// TIA Portal project "openness_project" (V17)

(* hardware
DEVICE "S71500/ET200MP station_1"  S7-1500 station
   slot 0: "Rail_0"  Rack  6ES7 590-1***0-0AA0
   slot 1: "N0001-S1-MC1.CC1-K30001"  CPU 1515F-2 PN  6ES7 515-2FM01-0AB0  V2.8
      slot 3: "CPU display_1"  6ES7591-1BA00-0AA0
      slot 32768: "PROFINET interface_1"  X1
         slot 32769: "Port_1"  X1 P1
         slot 32770: "Port_2"  X1 P2
      slot 33024: "PROFINET interface_2"  X2
         slot 33025: "Port_1"  X2 P1
      slot 34817: "Virtual CP interface port_1"  Virtual CP interface port  Virtual CP interface port
DEVICE "ET 200SP station_1"  ET 200SP-Station
   slot 0: "Rack_0"  Rack  6ES5 710-8MAx1
   slot 0: "IO device_1"  IM 155-6 PN ST  6ES7 155-6AU00-0BN0  V3.3
   slot 1: "DI 16x24VDC ST_1"  DI 16x24VDC ST  6ES7 131-6BH01-0BA0  V0.0
      slot 1: "DI 16x24VDC ST_1"  DI 16x24VDC ST
   slot 2: "F-DI 8x24VDC HF_1"  F-DI 8x24VDC HF  6ES7 136-6BA00-0CA0  V1.0
      slot 1: "F-DI 8x24VDC HF_1"  F-DI 8x24VDC HF
   slot 3: "F-DQ 4x24VDC/2A PM HF_1"  F-DQ 4x24VDC/2A PM HF  6ES7 136-6DB00-0CA0  V2.0
      slot 1: "F-DQ 4x24VDC/2A PM HF_1"  F-DQ 4x24VDC/2A PM HF
   slot 4: "DQ 16x24VDC/0.5A ST_1"  DQ 16x24VDC/0.5A ST  6ES7 132-6BH01-0BA0  V0.0
      slot 1: "DQ 16x24VDC/0.5A ST_1"  DQ 16x24VDC/0.5A ST
   slot 5: "CM 4xIO-Link_1"  CM 4xIO-Link  6ES7 137-6BD00-0BA0  V2.2
      slot 1: "CM 4xIO-Link_1"  6ES7 137-6BD00-0BA0
   slot 127: "BA 2xRJ45"  BA 2xRJ45  6ES7 193-6AR00-0AA0  V0.0
      slot 1: "Port_1"  X1 P1 R  6ES7 193-6AR00-0AA0  V0.0
      slot 2: "Port_2"  X1 P2 R  6ES7 193-6AR00-0AA0  V0.0
DEVICE "PNPN Coupler"  PnPn.Device
   slot 0: "Rack"  Rail  1.0
   slot 0: "PNPN Coupler.X1"  PN/PN Coupler  6ES7 158-3AD10-0XA0  V4.2
   slot 1: "PNPN Coupler.X2"  PN/PN Coupler  6ES7 158-3AD10-0XA0  V4.2
   slot 127: "BA 2xRJ45"  BA 2xRJ45  6ES7 193-6AR00-0AA0  V0.0
      slot 1: "Port_1"  X1 P1 R  6ES7 193-6AR00-0AA0  V0.0
      slot 2: "Port_2"  X1 P2 R  6ES7 193-6AR00-0AA0  V0.0
   slot 127: "BA 2xRJ45"  BA 2xRJ45  6ES7 193-6AR00-0AA0  V0.0
      slot 1: "Port_1"  X2 P1 R  6ES7 193-6AR00-0AA0  V0.0
      slot 2: "Port_2"  X2 P2 R  6ES7 193-6AR00-0AA0  V0.0
*)

// ===== PLC "N0001-S1-MC1.CC1-K30001"  CPU 1515F-2 PN =====
// protected blocks, not shown: "PNDD_IL_Diag_V1_11"

VAR_GLOBAL   // PLC tag table "Default tag table"
   "Tag_1" AT %Q10002.0 : Bool;
   "Tag_2" AT %Q100.0 : Bool;
   "System_Byte" AT %MB1 : Byte;
   "FirstScan" AT %M1.0 : Bool;
   "DiagStatusUpdate" AT %M1.1 : Bool;
   "AlwaysTRUE" AT %M1.2 : Bool;
   "AlwaysFALSE" AT %M1.3 : Bool;
   "Clock_Byte" AT %MB0 : Byte;
   "Clock_10Hz" AT %M0.0 : Bool;
   "Clock_5Hz" AT %M0.1 : Bool;
   "Clock_2.5Hz" AT %M0.2 : Bool;
   "Clock_2Hz" AT %M0.3 : Bool;
   "Clock_1.25Hz" AT %M0.4 : Bool;
   "Clock_1Hz" AT %M0.5 : Bool;
   "Clock_0.625Hz" AT %M0.6 : Bool;
   "Clock_0.5Hz" AT %M0.7 : Bool;
   "Tag_3" AT %Q0.0 : Bool;
   "Tag_4" AT %Q10002.1 : Bool;
   "Tag_5" AT %Q10002.2 : Bool;
   "Tag_6" AT %Q10005.0 : Bool;
   "!!FEEDBACK_INPUT_TAG_2!!" AT %I20.0 : Bool;
   "!!QBAD_INPUT_TAG_2!!" AT %I30.0 : Bool;
   "!!OUTPUT_CONTACTOR_TAG_2!!" AT %Q20.0 : Bool;
   "!!FEEDBACK_INPUT_TAG_1!!" AT %I200.0 : Bool;
   "!!QBAD_INPUT_TAG_1!!" AT %I300.0 : Bool;
   "!!OUTPUT_CONTACTOR_TAG_1!!" AT %Q200.0 : Bool;
   "FEEDBACK_INPUT_TAG_2" AT %I200.1 : Bool;
   "QBAD_INPUT_TAG_2" AT %I200.2 : Bool;
   "OUTPUT_CONTACTOR_TAG_2" AT %Q200.3 : Bool;
   "FEEDBACK_INPUT_TAG_1" AT %I200.4 : Bool;
   "QBAD_INPUT_TAG_1" AT %I200.5 : Bool;
   "OUTPUT_CONTACTOR_TAG_1" AT %Q200.6 : Bool;
   "FEEDBACK_INPUT_TAG_3" AT %I200.7 : Bool;
   "QBAD_INPUT_TAG_3" AT %I201.0 : Bool;
   "OUTPUT_CONTACTOR_TAG_3" AT %Q201.1 : Bool;
END_VAR

TYPE "SORTER_SPEED_STATE"
   STRUCT
      SORTER_STOPPED : Bool;
      ENCODER_BROKEN : Bool;
   END_STRUCT;
END_TYPE

TYPE "SLS_DATA"
   STRUCT
      PH1_RE : Bool;
      PH1_FE : Bool;
      PH2_RE : Bool;
      PH2_FE : Bool;
      PH1_ET : Time;
      PH2_ET : Time;
   END_STRUCT;
END_TYPE

DATA_BLOCK "Main_Safety_RTG1_DB"   // DB1, F_DB
{ S7_Optimized_Access := 'TRUE' }
NAME : FUSI
VERSION : 0.1
// stored: InstanceOfName Main_Safety_RTG1
"Main_Safety_RTG1"
BEGIN
END_DATA_BLOCK

DATA_BLOCK "00_Commissioning"   // DB2, F_DB
{ S7_Optimized_Access := 'TRUE' }
VERSION : 0.1
   VAR
      N0001_BYPASS_EXAMPLE : Bool;
   END_VAR
BEGIN
END_DATA_BLOCK

DATA_BLOCK "01_PushButton"   // DB3, F_DB
{ S7_Optimized_Access := 'TRUE' }
VERSION : 0.1
   VAR
      EXAMPLE_PushButton : Bool;
      EXAMPLE_PushButton_1 : Bool;
   END_VAR
BEGIN
END_DATA_BLOCK

DATA_BLOCK "02_COM"   // DB4, F_DB
{ S7_Optimized_Access := 'TRUE' }
VERSION : 0.1
   VAR
      EXAMPLE_SORTER_PB : Bool;
      EXAMPLE_SORTER_FDB : Bool;
      EXAMPLE_ZONE3_PB : Bool;
      EXAMPLE_ZONE3_FDB : Bool;
   END_VAR
BEGIN
END_DATA_BLOCK

DATA_BLOCK "03_FDBACK"   // DB5, F_DB
{ S7_Optimized_Access := 'TRUE' }
VERSION : 0.1
   VAR
      EXAMPLE_FDBACK : Bool;
      EXAMPLE_FDBACK_SORTER : Bool;
      EXAMPLE_FDBACK_DU : Bool;
      EXAMPLE_FDBACK_ISPC : Bool;
   END_VAR
BEGIN
END_DATA_BLOCK

DATA_BLOCK "04_SPEED"   // DB6, F_DB
{ S7_Optimized_Access := 'TRUE' }
VERSION : 0.1
   VAR
      SLS_DATA_SORTER1 : "SLS_DATA";
   END_VAR
BEGIN
END_DATA_BLOCK

DATA_BLOCK "05_EM_STATE"   // DB7, F_DB
{ S7_Optimized_Access := 'TRUE' }
VERSION : 0.1
   VAR
      RESET : Bool;
      EM_SORTER : Bool;
      EM_ZONE_EXAMPLE : Bool;
      SORTER_STOP : Bool;
      POWER_CUT_SORTER : Bool;
      SAFETY_BREAKER_COM : Bool;
      DOOR_COM : Bool;
      DOOR_ALARM_EXAMPLE : Bool;
      N_TRIG_RESET : Bool;
      "!!RESET_CONDITION_2!!" : Bool;
      "!!ON_CONDITION_2!!" : Bool;
      "!!RESET_CONDITION_1!!" : Bool;
      "!!ON_CONDITION_1!!" : Bool;
      ON_CONDITION_1 : Bool;
      RESET_CONDITION_1 : Bool;
      ON_CONDITION_2 : Bool;
      RESET_CONDITION_2 : Bool;
      ON_CONDITION_3 : Bool;
      RESET_CONDITION_3 : Bool;
   END_VAR
BEGIN
END_DATA_BLOCK

DATA_BLOCK "06_Settings"   // DB8, F_DB
{ S7_Optimized_Access := 'TRUE' }
VERSION : 0.1
   VAR
      Tristate : Bool;
   END_VAR
BEGIN
END_DATA_BLOCK

DATA_BLOCK "Speed_Control_SLS_DB"   // DB22, F_DB
{ S7_Optimized_Access := 'TRUE' }
VERSION : 0.1
// stored: InstanceOfName 01_Speed_Control_SLS
"01_Speed_Control_SLS"
BEGIN
END_DATA_BLOCK

DATA_BLOCK "08_AL_FILTER"   // DB25
{ S7_Optimized_Access := 'TRUE' }
VERSION : 0.1
   VAR
      "N0001-EXAMPLE" : Bool;
   END_VAR
BEGIN
END_DATA_BLOCK

DATA_BLOCK "00_Diagnostic_Profinet_DB"   // DB43
{ S7_Optimized_Access := 'TRUE' }
VERSION : 0.1
   VAR
      "Local~PROFINET_EXAMPLE" : Array[0..1023] of Bool;   // one array per subnet
   END_VAR
BEGIN
END_DATA_BLOCK

DATA_BLOCK "07_DOOR"   // DB48, F_DB
{ S7_Optimized_Access := 'TRUE' }
VERSION : 0.1
   VAR
      MAINT_D1_EM : Bool;
      MAINT_D2_EM : Bool;
   END_VAR
BEGIN
END_DATA_BLOCK

// folder: 00_PushButton

DATA_BLOCK "N0001-EXAMPLE-01"   // DB9, F_DB
{ S7_Optimized_Access := 'TRUE' }
VERSION : 0.1
// stored: InstanceOfName 00_Push-Button_Input
"00_Push-Button_Input"
BEGIN
END_DATA_BLOCK

// folder: 01_Feedback error

DATA_BLOCK "FDBACK error_EXAMPLE"   // DB16, F_DB
{ S7_Optimized_Access := 'TRUE' }
VERSION : 0.1
// stored: InstanceOfName 03_FDBACK error
"03_FDBACK error"
BEGIN
END_DATA_BLOCK

DATA_BLOCK "FDBACK-N0001-1"   // DB19, F_DB
{ S7_Optimized_Access := 'TRUE' }
VERSION : 0.1
// stored: InstanceOfName 03_FDBACK error
"03_FDBACK error"
BEGIN
END_DATA_BLOCK

// folder: 02_Speed Control

DATA_BLOCK "Speed_Control_DB"   // DB17, F_DB
{ S7_Optimized_Access := 'TRUE' }
VERSION : 0.1
// stored: InstanceOfName 01_Speed_Control
"01_Speed_Control"
BEGIN
END_DATA_BLOCK

// folder: 03_Gate manager

DATA_BLOCK "MAINT_DOOR1"   // DB21, F_DB
{ S7_Optimized_Access := 'TRUE' }
VERSION : 0.1
// stored: InstanceOfName 02_Safety_Door
"02_Safety_Door"
BEGIN
END_DATA_BLOCK

// folder: (top level)

FUNCTION_BLOCK "Main_Safety_RTG1"   // FB1, F_FBD
{ S7_Optimized_Access := 'TRUE' }
   VAR_TEMP
      t_Reset : Bool;
   END_VAR
   VAR_TEMP   // added for the SCL form of the ladder/FBD networks
      _w1 : Bool;
      _w2 : Bool;
   END_VAR
BEGIN

REGION Network 1: For commissioning
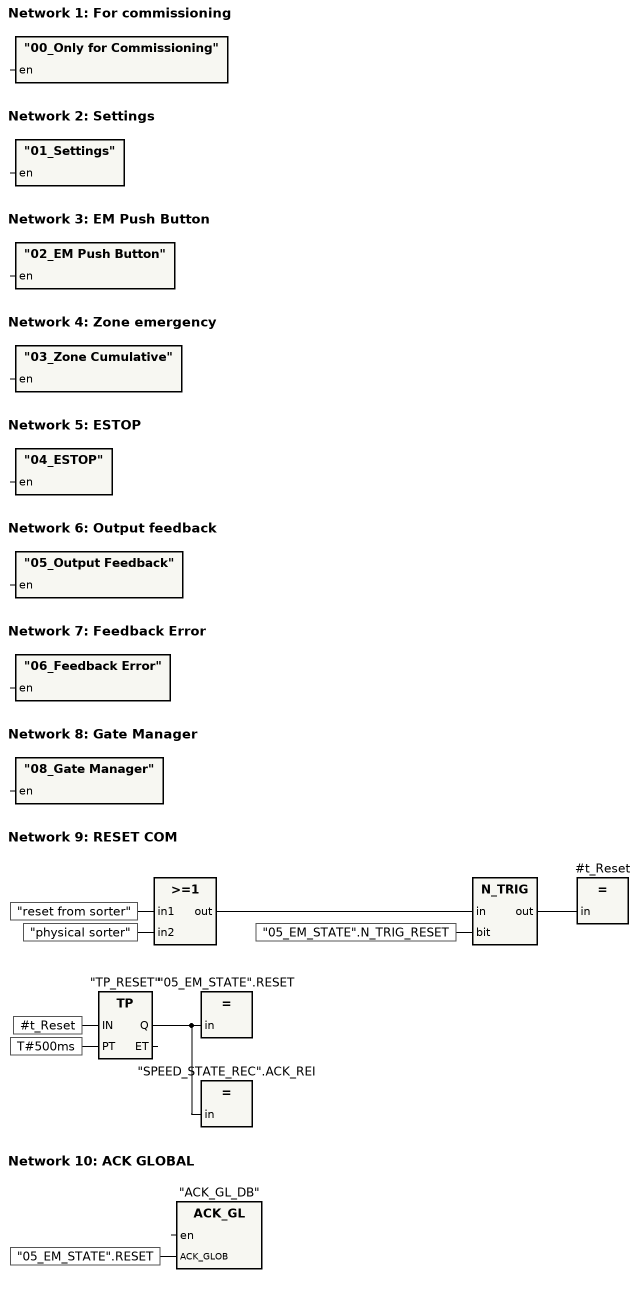
   "00_Only for Commissioning"();
END_REGION

REGION Network 2: Settings
   "01_Settings"();
END_REGION

REGION Network 3: EM Push Button
   "02_EM Push Button"();
END_REGION

REGION Network 4: Zone emergency
   "03_Zone Cumulative"();
END_REGION

REGION Network 5: ESTOP
   "04_ESTOP"();
END_REGION

REGION Network 6: Output feedback
   "05_Output Feedback"();
END_REGION

REGION Network 7: Feedback Error
   "06_Feedback Error"();
END_REGION

REGION Network 8: Gate Manager
   "08_Gate Manager"();
END_REGION

REGION Network 9: RESET COM
   // Add any other reset
   #_w1 := "reset from sorter" OR "physical sorter";
   #_w2 := NOT #_w1 AND "05_EM_STATE".N_TRIG_RESET;   // falling edge
   "05_EM_STATE".N_TRIG_RESET := #_w1;
   #t_Reset := #_w2;
   "TP_RESET".TP(IN := #t_Reset, PT := T#500ms);
   "05_EM_STATE".RESET := "TP_RESET".Q;
   "SPEED_STATE_REC".ACK_REI := "TP_RESET".Q;
END_REGION

REGION Network 10: ACK GLOBAL
   "ACK_GL_DB"(ACK_GLOB := "05_EM_STATE".RESET);   // ACK_GL
END_REGION
END_FUNCTION_BLOCK

FUNCTION_BLOCK "00_Push-Button_Input"   // FB2, F_LAD
TITLE = Push-Button_Input_ET200
{ S7_Optimized_Access := 'TRUE' }
VERSION : 0.1
// Input
// Bypass_ET200
// IN_1
// IN_2
// IN_3
// IN_4
// ON_Diag
// ON_Lamp
// Reset
// Output
// OUT_1
// OUT_2
// OUT_3
// OUT_4
// Diag_1
// Diag_2
// Diag_3
// Diag_4
// Lamp_1
// Lamp_2
// Lamp_3
// Lamp_4
// 
// InOut
// 
// Static
// ESTOP_1
// ESTOP_2
// ESTOP_3
// ESTOP_4
// Temp
// 
// Constant
   VAR_INPUT
      Bypass_ET200 : Bool;
      IN_1 : Bool;
      IN_2 : Bool;
      IN_3 : Bool;
      IN_4 : Bool;
      ON_Tristate : Bool;
      ON_Lamp : Bool;
      Reset : Bool;
      REAC_DELAY : Time;   // Reactivation delay= the OUT goes from 0 to 1 after this time
   END_VAR
   VAR_OUTPUT
      OUT_1 : Bool;
      OUT_2 : Bool;
      OUT_3 : Bool;
      OUT_4 : Bool;
      Diag_1 : Bool;
      Diag_2 : Bool;
      Diag_3 : Bool;
      Diag_4 : Bool;
      Lamp_1 : Bool;
      Lamp_2 : Bool;
      Lamp_3 : Bool;
      Lamp_4 : Bool;
   END_VAR
   VAR
      ESTOP_1 : ESTOP1;
      ESTOP_2 : ESTOP1;
      ESTOP_3 : ESTOP1;
      ESTOP_4 : ESTOP1;
      TON_1 : TON;
      TON_2 : TON;
      TON_3 : TON;
      TON_4 : TON;
   END_VAR
BEGIN

REGION Network 1 (F_FBD): Card: 4 Input safety for Push-Button
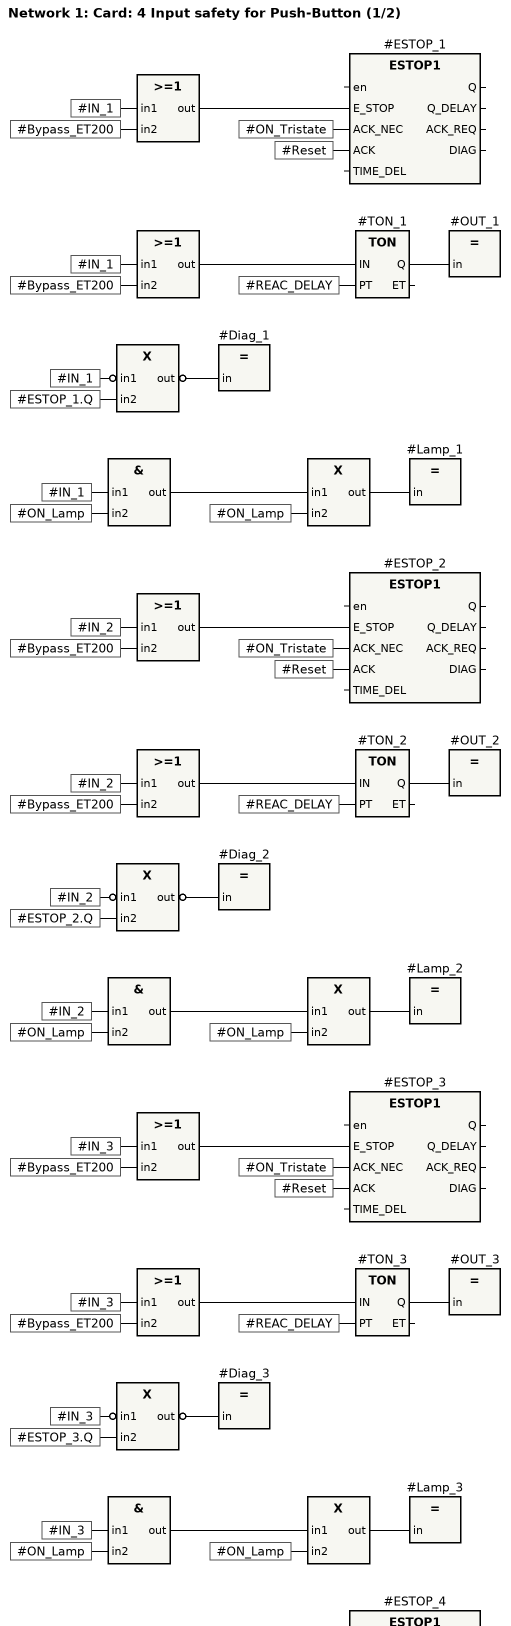
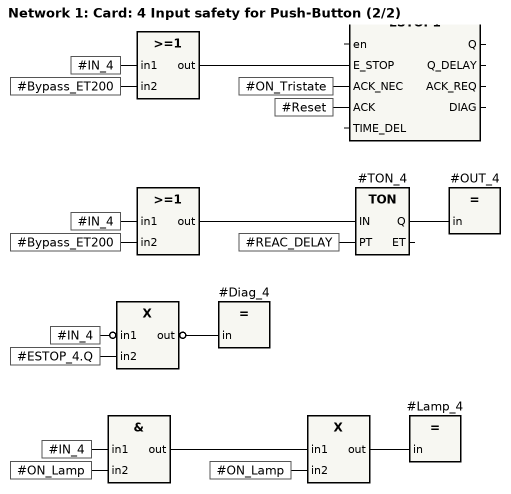
   #ESTOP_1(E_STOP := #IN_1 OR #Bypass_ET200, ACK_NEC := #ON_Tristate, ACK := #Reset);   // ESTOP1
   #TON_1.TON(IN := #IN_1 OR #Bypass_ET200, PT := #REAC_DELAY);
   #OUT_1 := #TON_1.Q;
   #Diag_1 := NOT (NOT #IN_1 XOR #ESTOP_1.Q);
   #Lamp_1 := (#IN_1 AND #ON_Lamp) XOR #ON_Lamp;
   #ESTOP_2(E_STOP := #IN_2 OR #Bypass_ET200, ACK_NEC := #ON_Tristate, ACK := #Reset);   // ESTOP1
   #TON_2.TON(IN := #IN_2 OR #Bypass_ET200, PT := #REAC_DELAY);
   #OUT_2 := #TON_2.Q;
   #Diag_2 := NOT (NOT #IN_2 XOR #ESTOP_2.Q);
   #Lamp_2 := (#IN_2 AND #ON_Lamp) XOR #ON_Lamp;
   #ESTOP_3(E_STOP := #IN_3 OR #Bypass_ET200, ACK_NEC := #ON_Tristate, ACK := #Reset);   // ESTOP1
   #TON_3.TON(IN := #IN_3 OR #Bypass_ET200, PT := #REAC_DELAY);
   #OUT_3 := #TON_3.Q;
   #Diag_3 := NOT (NOT #IN_3 XOR #ESTOP_3.Q);
   #Lamp_3 := (#IN_3 AND #ON_Lamp) XOR #ON_Lamp;
   #ESTOP_4(E_STOP := #IN_4 OR #Bypass_ET200, ACK_NEC := #ON_Tristate, ACK := #Reset);   // ESTOP1
   #TON_4.TON(IN := #IN_4 OR #Bypass_ET200, PT := #REAC_DELAY);
   #OUT_4 := #TON_4.Q;
   #Diag_4 := NOT (NOT #IN_4 XOR #ESTOP_4.Q);
   #Lamp_4 := (#IN_4 AND #ON_Lamp) XOR #ON_Lamp;
END_REGION
END_FUNCTION_BLOCK

FUNCTION_BLOCK "01_Speed_Control"   // FB3, F_FBD
{ S7_Optimized_Access := 'TRUE' }
VERSION : 0.1
   VAR_INPUT
      "Sorter in RUN" : Bool;   // Sorter in Run from sorter
      PH1 : Bool;   // Phisycal input PH1
      PH2 : Bool;   // Phisycal input PH2
      "Time" : Time := T#4s;   // Time used to check the state of the sorter
      Running_Delay : Time := T#5s;   // Delay to sorter running
   END_VAR
   VAR_OUTPUT
      "Sorter STOP" : Bool;
      "Broken PH safety encoder" : Bool;
      "Stop PH1" : Bool;
      "Stop PH2" : Bool;
      "Broken PH1" : Bool;
      "Broken PH2" : Bool;
   END_VAR
   VAR
      TON_Stop1_PH1 : TON;
      TON_Stop2_PH1 : TON;
      TON_Broken1_PH1 : TON;
      TON_Broken2_PH1 : TON;
      TON_Stop1_PH2 : TON;
      TON_Stop2_PH2 : TON;
      TON_Broken1_PH2 : TON;
      TON_Broken2_PH2 : TON;
      TON_SORTER_DELAY : TON;
   END_VAR
   VAR_TEMP
      "t_Stop PH1_temp" : Bool;
      "t_Stop PH2_temp" : Bool;
      "t_Broken PH1_temp" : Bool;
      "t_Broken PH2_temp" : Bool;
      t_Sorter_Running : Bool;
   END_VAR
   VAR_TEMP   // added for the SCL form of the ladder/FBD networks
      _w1 : Bool;
   END_VAR
BEGIN

REGION Network 1
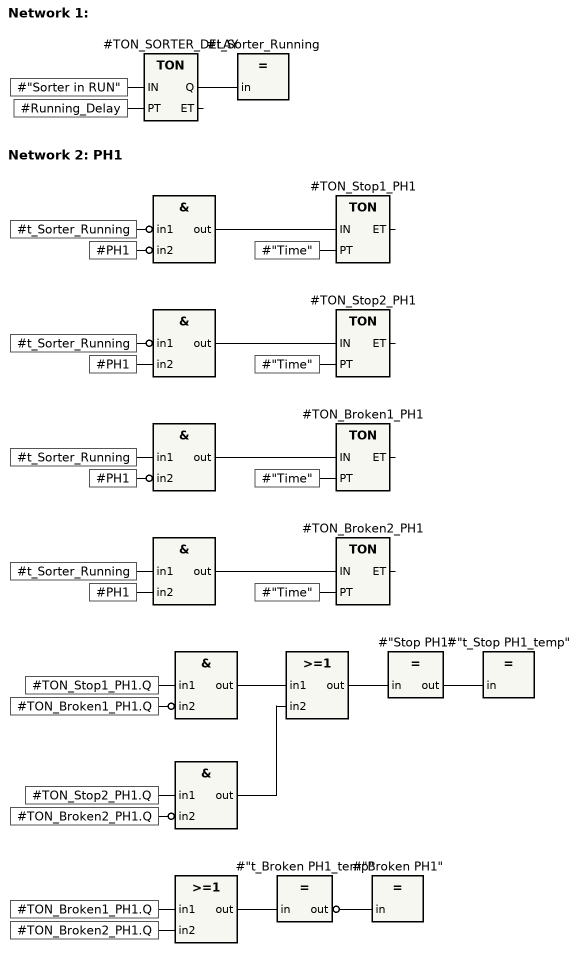
   #TON_SORTER_DELAY.TON(IN := #"Sorter in RUN", PT := #Running_Delay);
   #t_Sorter_Running := #TON_SORTER_DELAY.Q;
END_REGION

REGION Network 2: PH1
   #TON_Stop1_PH1.TON(IN := NOT #t_Sorter_Running AND NOT #PH1, PT := #"Time");
   #TON_Stop2_PH1.TON(IN := NOT #t_Sorter_Running AND #PH1, PT := #"Time");
   #TON_Broken1_PH1.TON(IN := #t_Sorter_Running AND NOT #PH1, PT := #"Time");
   #TON_Broken2_PH1.TON(IN := #t_Sorter_Running AND #PH1, PT := #"Time");
   #"Stop PH1" := (#TON_Stop1_PH1.Q AND NOT #TON_Broken1_PH1.Q) OR (#TON_Stop2_PH1.Q AND NOT #TON_Broken2_PH1.Q);
   #"t_Stop PH1_temp" := #"Stop PH1";
   #_w1 := #TON_Broken1_PH1.Q OR #TON_Broken2_PH1.Q;
   #"t_Broken PH1_temp" := #_w1;
   #"Broken PH1" := NOT #_w1;
END_REGION

REGION Network 3: PH2
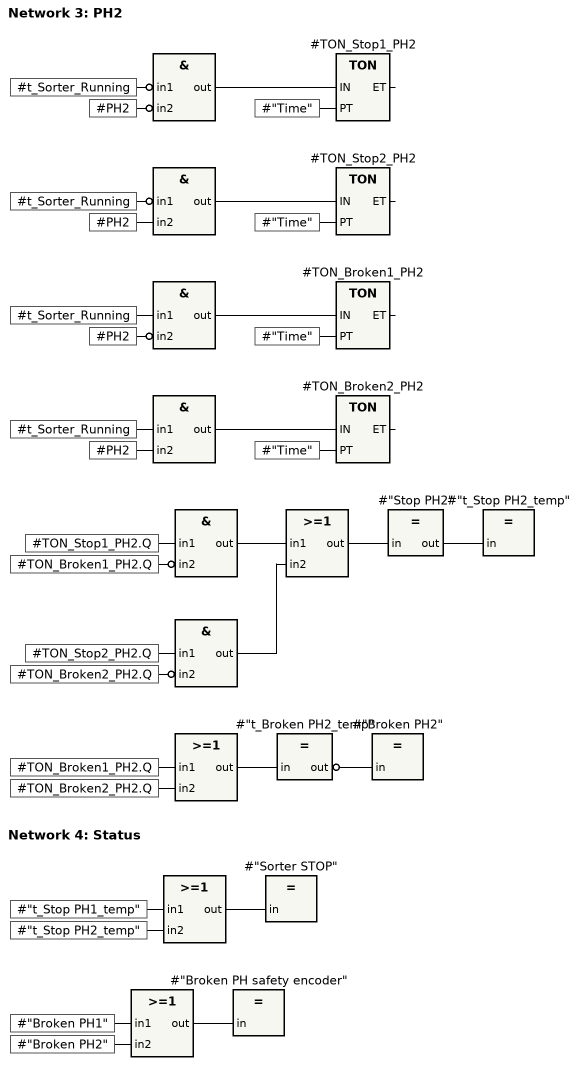
   #TON_Stop1_PH2.TON(IN := NOT #t_Sorter_Running AND NOT #PH2, PT := #"Time");
   #TON_Stop2_PH2.TON(IN := NOT #t_Sorter_Running AND #PH2, PT := #"Time");
   #TON_Broken1_PH2.TON(IN := #t_Sorter_Running AND NOT #PH2, PT := #"Time");
   #TON_Broken2_PH2.TON(IN := #t_Sorter_Running AND #PH2, PT := #"Time");
   #"Stop PH2" := (#TON_Stop1_PH2.Q AND NOT #TON_Broken1_PH2.Q) OR (#TON_Stop2_PH2.Q AND NOT #TON_Broken2_PH2.Q);
   #"t_Stop PH2_temp" := #"Stop PH2";
   #_w1 := #TON_Broken1_PH2.Q OR #TON_Broken2_PH2.Q;
   #"t_Broken PH2_temp" := #_w1;
   #"Broken PH2" := NOT #_w1;
END_REGION

REGION Network 4: Status
   #"Sorter STOP" := #"t_Stop PH1_temp" OR #"t_Stop PH2_temp";
   #"Broken PH safety encoder" := #"Broken PH1" OR #"Broken PH2";
END_REGION
END_FUNCTION_BLOCK

FUNCTION_BLOCK "03_FDBACK error"   // FB4, F_LAD
TITLE = 03_FDBACK error
{ S7_Optimized_Access := 'TRUE' }
VERSION : 0.1
// Input
// Commissioning_bypass
// FDBACK ERROR 1
// FDBACK ERROR 2
// FDBACK ERROR 3
// FDBACK ERROR 4
// FDBACK ERROR 5
// FDBACK ERROR 6
// FDBACK ERROR 7
// FDBACK ERROR 8
// FDBACK ERROR 9
// FDBACK ERROR 10
// 
// Output
// Cumulative FDBACK
// 
// InOut
// 
// Static
// 
// Temp
// 
// Constant
   VAR_INPUT
      Commissioning_bypass : Bool;
      "FDBACK ERROR 1" : Bool;
      "FDBACK ERROR 2" : Bool;
      "FDBACK ERROR 3" : Bool;
      "FDBACK ERROR 4" : Bool;
      "FDBACK ERROR 5" : Bool;
      "FDBACK ERROR 6" : Bool;
      "FDBACK ERROR 7" : Bool;
      "FDBACK ERROR 8" : Bool;
   END_VAR
   VAR_OUTPUT
      "Cumulative FDBACK" : Bool;
      "ERROR 1" : Bool;
      "ERROR 2" : Bool;
      "ERROR 3" : Bool;
      "ERROR 4" : Bool;
      "ERROR 5" : Bool;
      "ERROR 6" : Bool;
      "ERROR 7" : Bool;
      "ERROR 8" : Bool;
   END_VAR
BEGIN

REGION Network 1: First channel
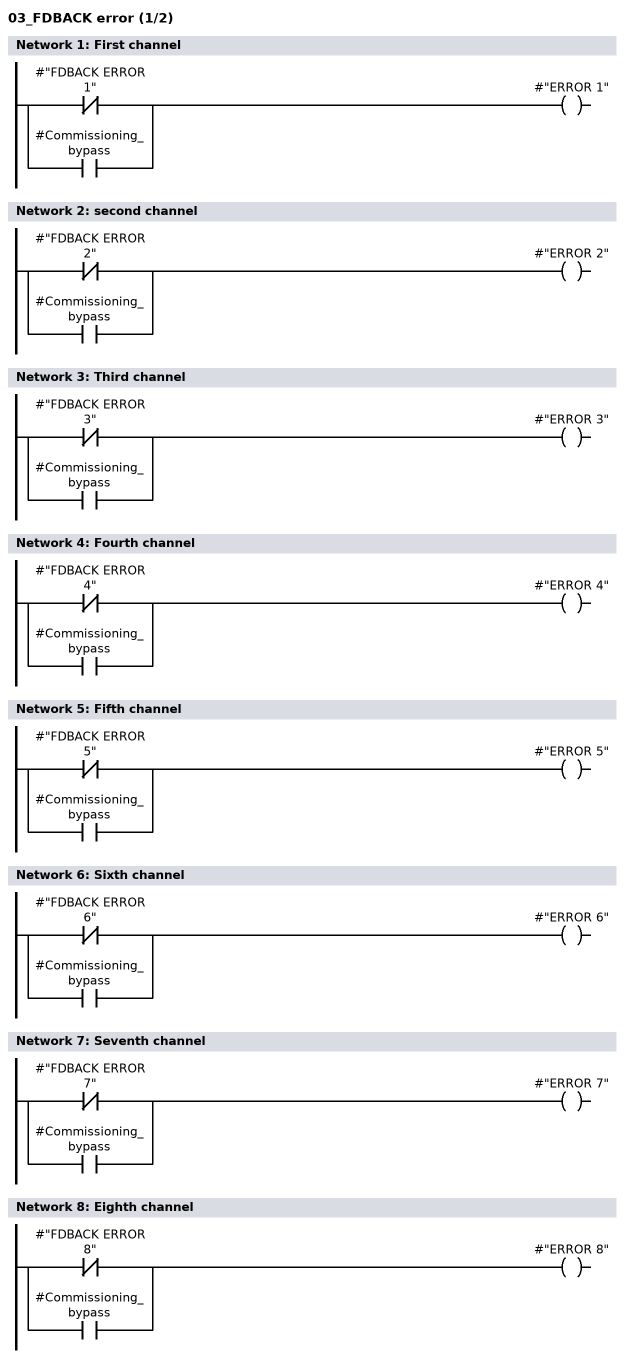
   RUNG wire#powerrail
      I_Contact( #"FDBACK ERROR 1" )
      wire#w1
      Coil( #"ERROR 1" )
   END_RUNG
   RUNG wire#powerrail
      Contact( #Commissioning_bypass )
   END_RUNG wire#w1
   // the same network as SCL:
   #"ERROR 1" := NOT #"FDBACK ERROR 1" OR #Commissioning_bypass;
END_REGION

REGION Network 2: second channel
   RUNG wire#powerrail
      I_Contact( #"FDBACK ERROR 2" )
      wire#w1
      Coil( #"ERROR 2" )
   END_RUNG
   RUNG wire#powerrail
      Contact( #Commissioning_bypass )
   END_RUNG wire#w1
   // the same network as SCL:
   #"ERROR 2" := NOT #"FDBACK ERROR 2" OR #Commissioning_bypass;
END_REGION

REGION Network 3: Third channel
   RUNG wire#powerrail
      I_Contact( #"FDBACK ERROR 3" )
      wire#w1
      Coil( #"ERROR 3" )
   END_RUNG
   RUNG wire#powerrail
      Contact( #Commissioning_bypass )
   END_RUNG wire#w1
   // the same network as SCL:
   #"ERROR 3" := NOT #"FDBACK ERROR 3" OR #Commissioning_bypass;
END_REGION

REGION Network 4: Fourth channel
   RUNG wire#powerrail
      I_Contact( #"FDBACK ERROR 4" )
      wire#w1
      Coil( #"ERROR 4" )
   END_RUNG
   RUNG wire#powerrail
      Contact( #Commissioning_bypass )
   END_RUNG wire#w1
   // the same network as SCL:
   #"ERROR 4" := NOT #"FDBACK ERROR 4" OR #Commissioning_bypass;
END_REGION

REGION Network 5: Fifth channel
   RUNG wire#powerrail
      I_Contact( #"FDBACK ERROR 5" )
      wire#w1
      Coil( #"ERROR 5" )
   END_RUNG
   RUNG wire#powerrail
      Contact( #Commissioning_bypass )
   END_RUNG wire#w1
   // the same network as SCL:
   #"ERROR 5" := NOT #"FDBACK ERROR 5" OR #Commissioning_bypass;
END_REGION

REGION Network 6: Sixth channel
   RUNG wire#powerrail
      I_Contact( #"FDBACK ERROR 6" )
      wire#w1
      Coil( #"ERROR 6" )
   END_RUNG
   RUNG wire#powerrail
      Contact( #Commissioning_bypass )
   END_RUNG wire#w1
   // the same network as SCL:
   #"ERROR 6" := NOT #"FDBACK ERROR 6" OR #Commissioning_bypass;
END_REGION

REGION Network 7: Seventh channel
   RUNG wire#powerrail
      I_Contact( #"FDBACK ERROR 7" )
      wire#w1
      Coil( #"ERROR 7" )
   END_RUNG
   RUNG wire#powerrail
      Contact( #Commissioning_bypass )
   END_RUNG wire#w1
   // the same network as SCL:
   #"ERROR 7" := NOT #"FDBACK ERROR 7" OR #Commissioning_bypass;
END_REGION

REGION Network 8: Eighth channel
   RUNG wire#powerrail
      I_Contact( #"FDBACK ERROR 8" )
      wire#w1
      Coil( #"ERROR 8" )
   END_RUNG
   RUNG wire#powerrail
      Contact( #Commissioning_bypass )
   END_RUNG wire#w1
   // the same network as SCL:
   #"ERROR 8" := NOT #"FDBACK ERROR 8" OR #Commissioning_bypass;
END_REGION

REGION Network 9: Cumulative error
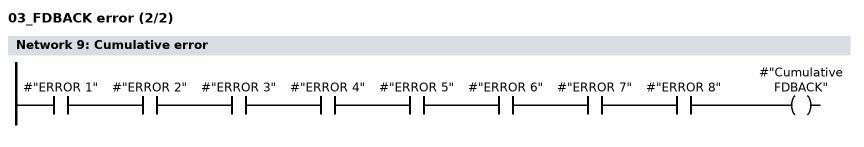
   RUNG wire#powerrail
      Contact( #"ERROR 1" )
      Contact( #"ERROR 2" )
      Contact( #"ERROR 3" )
      Contact( #"ERROR 4" )
      Contact( #"ERROR 5" )
      Contact( #"ERROR 6" )
      Contact( #"ERROR 7" )
      Contact( #"ERROR 8" )
      Coil( #"Cumulative FDBACK" )
   END_RUNG
   // the same network as SCL:
   #"Cumulative FDBACK" := #"ERROR 1" AND #"ERROR 2" AND #"ERROR 3" AND #"ERROR 4" AND #"ERROR 5" AND #"ERROR 6" AND #"ERROR 7" AND #"ERROR 8";
END_REGION
END_FUNCTION_BLOCK

FUNCTION_BLOCK "02_Safety_Door"   // FB5, F_LAD
{ S7_Optimized_Access := 'TRUE' }
VERSION : 0.1
   VAR_INPUT
      Bypass_For_Commissioning : Bool;
      DIAG : Bool := TRUE;
      CH1 : Bool := TRUE;
      CH2 : Bool := TRUE;
      "Sorter_Running_from MSC" : Bool;
      Sorter_Stop_from_Encoder : Bool;
      Open_Request : Bool;
      Alarm_Filter : Bool;
      Sorter_Door : Bool := TRUE;   // If =1 sorter door management, if =0 management via ESTOP
      ACK_NEC : Bool;   // For non sorter doors
      ACK : Bool;   // For non sorter doors
   END_VAR
   VAR_OUTPUT
      Solenoid : Bool;
      EM_Cut : Bool;
      EM_Cut_Delay : Bool;
      Diag_Open : Bool;
      Diag_Alarm : Bool;
   END_VAR
   VAR
      "E-STOP" : ESTOP1;
      TON_Alarm : TON;
   END_VAR
   VAR_TEMP
      Alarm_Temp : Bool;
      t_ALARM : Bool;
   END_VAR
BEGIN

REGION Network 1: Emergency cut
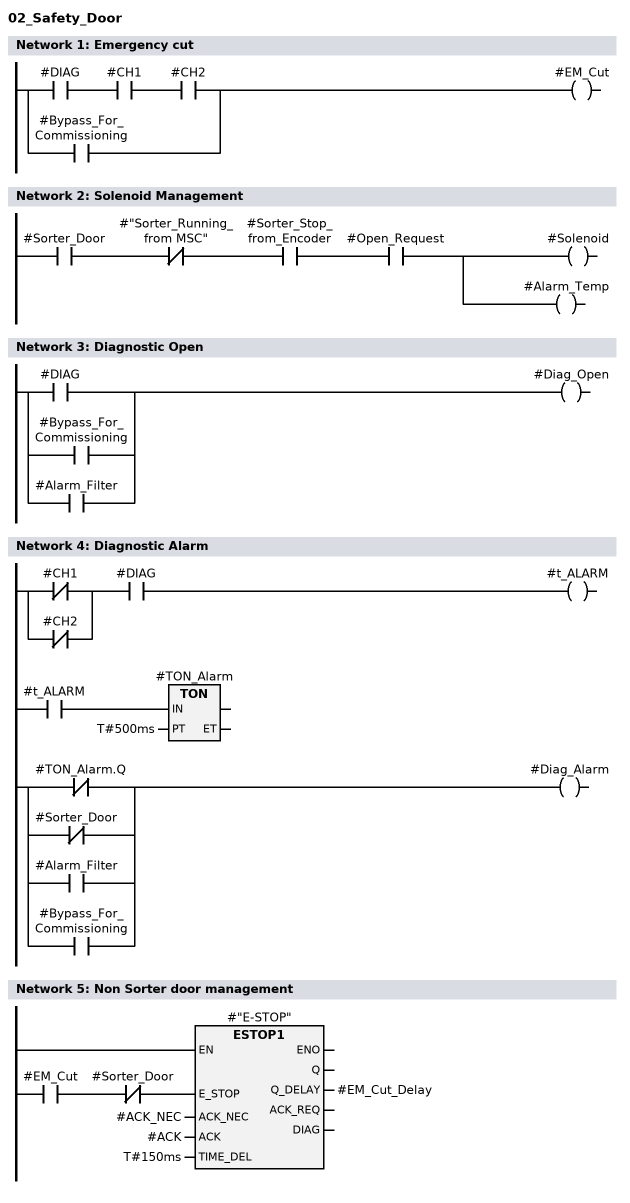
   RUNG wire#powerrail
      Contact( #DIAG )
      Contact( #CH1 )
      Contact( #CH2 )
      wire#w1
      Coil( #EM_Cut )
   END_RUNG
   RUNG wire#powerrail
      Contact( #Bypass_For_Commissioning )
   END_RUNG wire#w1
   // the same network as SCL:
   #EM_Cut := (#DIAG AND #CH1 AND #CH2) OR #Bypass_For_Commissioning;
END_REGION

REGION Network 2: Solenoid Management
   RUNG wire#powerrail
      Contact( #Sorter_Door )
      I_Contact( #"Sorter_Running_from MSC" )
      Contact( #Sorter_Stop_from_Encoder )
      Contact( #Open_Request )
      wire#w1
      Coil( #Solenoid )
   END_RUNG
   RUNG wire#w1
      Coil( #Alarm_Temp )
   END_RUNG
   // the same network as SCL:
   #Solenoid := #Sorter_Door AND NOT #"Sorter_Running_from MSC" AND #Sorter_Stop_from_Encoder AND #Open_Request;
   #Alarm_Temp := #Solenoid;
END_REGION

REGION Network 3: Diagnostic Open
   RUNG wire#powerrail
      Contact( #DIAG )
      wire#w1
      Coil( #Diag_Open )
   END_RUNG
   RUNG wire#powerrail
      Contact( #Bypass_For_Commissioning )
   END_RUNG wire#w1
   RUNG wire#powerrail
      Contact( #Alarm_Filter )
   END_RUNG wire#w1
   // the same network as SCL:
   #Diag_Open := #DIAG OR #Bypass_For_Commissioning OR #Alarm_Filter;
END_REGION

REGION Network 4: Diagnostic Alarm
   #t_ALARM := (NOT #CH1 OR NOT #CH2) AND #DIAG;
   #TON_Alarm.TON(IN := #t_ALARM, PT := T#500ms);
   #Diag_Alarm := NOT #TON_Alarm.Q OR NOT #Sorter_Door OR #Alarm_Filter OR #Bypass_For_Commissioning;
END_REGION

REGION Network 5: Non Sorter door management
   #"E-STOP"(E_STOP := #EM_Cut AND NOT #Sorter_Door,   // ESTOP1
             ACK_NEC := #ACK_NEC,
             ACK := #ACK,
             TIME_DEL := T#150ms,
             Q_DELAY => #EM_Cut_Delay);
END_REGION
END_FUNCTION_BLOCK

FUNCTION_BLOCK "01_Speed_Control_SLS"   // FB7, F_LAD
{ S7_Optimized_Access := 'TRUE' }
VERSION : 0.1
   VAR_INPUT
      PH1 : Bool;
      PH2 : Bool;
      SORTER_RUNNING_MSC : Bool;
      SLS_NOT_EN : Bool;
      "MIN[time]" : Time;   // SLS Limit[ms] = Blade length[mm] / Speed[mm/s]
      "MAX[time]" : Time := T#4s;   // Sorter not moving
      "DelayRunning[time]" : Time := T#5s;   // Delay running status from sorter
   END_VAR
   VAR_OUTPUT
      SPEED_ZERO : Bool;
      SPEED_TOOHIGH : Bool;
      "PH1 Broken" : Bool;
      "PH2 Broken" : Bool;
      ENC_BROKEN : Bool;
   END_VAR
   VAR_IN_OUT
      SLS_DATA : "SLS_DATA";
   END_VAR
   VAR
      Time_Limit : Time := T#10s;
      TON_SLS_T_PH1 : TON;
      TON_SLS_T_PH2 : TON;
      TOF_PH1_WORKING : TOF;
      TOF_PH2_WORKING : TOF;
      TON_SORTER_STOP : TON;
      TON_TIMEOUT_COUNT : TON;
      TON_DELAY_RUNNING_STATUS : TON;
      CTU_SLS_PH1 : CTU;
      CTU_SLS_PH2 : CTU;
   END_VAR
   VAR_TEMP
      t_SpeedTH_PH1 : Bool;
      t_SpeedTH_PH2 : Bool;
      t_Speed0_PH1 : Bool;
      t_Speed0_PH2 : Bool;
      t_PH1_FE : Bool;
      t_PH2_FE : Bool;
      t_PH1_RE : Bool;
      t_PH2_RE : Bool;
      t_PH1_BRK : Bool;
      t_PH2_BRK : Bool;
      t_SorterRunning : Bool;
   END_VAR
   VAR CONSTANT
      NUM_STH : Int := 3;   // Number of blades with speed too high in TIMEOUT_CTU time
      TIMEOUT_CTU : Time := T#5s;   // Deltatime to count number of blades too fast
   END_VAR
   VAR_TEMP   // added for the SCL form of the ladder/FBD networks
      _w1 : Bool;
      _w2 : Bool;
   END_VAR
BEGIN

REGION Network 1: Falling Edges
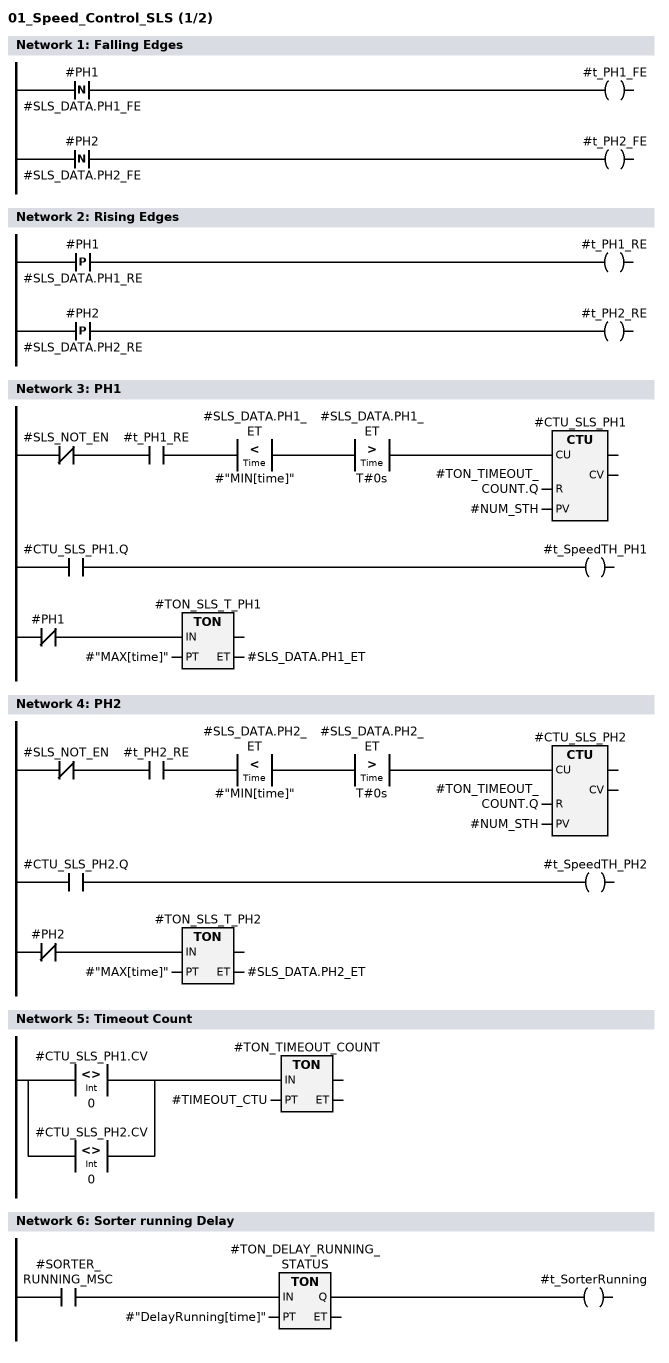
   RUNG wire#powerrail
      N_Contact(operand := #PH1, bit := #SLS_DATA.PH1_FE)
      Coil( #t_PH1_FE )
   END_RUNG
   RUNG wire#powerrail
      N_Contact(operand := #PH2, bit := #SLS_DATA.PH2_FE)
      Coil( #t_PH2_FE )
   END_RUNG
   // the same network as SCL:
   #_w1 := NOT #PH1 AND #SLS_DATA.PH1_FE;   // falling edge of #PH1
   #SLS_DATA.PH1_FE := #PH1;
   #t_PH1_FE := #_w1;
   #_w2 := NOT #PH2 AND #SLS_DATA.PH2_FE;   // falling edge of #PH2
   #SLS_DATA.PH2_FE := #PH2;
   #t_PH2_FE := #_w2;
END_REGION

REGION Network 2: Rising Edges
   RUNG wire#powerrail
      P_Contact(operand := #PH1, bit := #SLS_DATA.PH1_RE)
      Coil( #t_PH1_RE )
   END_RUNG
   RUNG wire#powerrail
      P_Contact(operand := #PH2, bit := #SLS_DATA.PH2_RE)
      Coil( #t_PH2_RE )
   END_RUNG
   // the same network as SCL:
   #_w1 := #PH1 AND NOT #SLS_DATA.PH1_RE;   // rising edge of #PH1
   #SLS_DATA.PH1_RE := #PH1;
   #t_PH1_RE := #_w1;
   #_w2 := #PH2 AND NOT #SLS_DATA.PH2_RE;   // rising edge of #PH2
   #SLS_DATA.PH2_RE := #PH2;
   #t_PH2_RE := #_w2;
END_REGION

REGION Network 3: PH1
   #CTU_SLS_PH1.CTU(CU := NOT #SLS_NOT_EN AND #t_PH1_RE AND (#SLS_DATA.PH1_ET < #"MIN[time]") AND (#SLS_DATA.PH1_ET > T#0s),
                    R := #TON_TIMEOUT_COUNT.Q,
                    PV := #NUM_STH);
   #t_SpeedTH_PH1 := #CTU_SLS_PH1.Q;
   #TON_SLS_T_PH1.TON(IN := NOT #PH1, PT := #"MAX[time]", ET => #SLS_DATA.PH1_ET);
END_REGION

REGION Network 4: PH2
   #CTU_SLS_PH2.CTU(CU := NOT #SLS_NOT_EN AND #t_PH2_RE AND (#SLS_DATA.PH2_ET < #"MIN[time]") AND (#SLS_DATA.PH2_ET > T#0s),
                    R := #TON_TIMEOUT_COUNT.Q,
                    PV := #NUM_STH);
   #t_SpeedTH_PH2 := #CTU_SLS_PH2.Q;
   #TON_SLS_T_PH2.TON(IN := NOT #PH2, PT := #"MAX[time]", ET => #SLS_DATA.PH2_ET);
END_REGION

REGION Network 5: Timeout Count
   #TON_TIMEOUT_COUNT.TON(IN := (#CTU_SLS_PH1.CV <> 0) OR (#CTU_SLS_PH2.CV <> 0), PT := #TIMEOUT_CTU);
END_REGION

REGION Network 6: Sorter running Delay
   #TON_DELAY_RUNNING_STATUS.TON(IN := #SORTER_RUNNING_MSC, PT := #"DelayRunning[time]");
   #t_SorterRunning := #TON_DELAY_RUNNING_STATUS.Q;
END_REGION

REGION Network 7: Speed too high
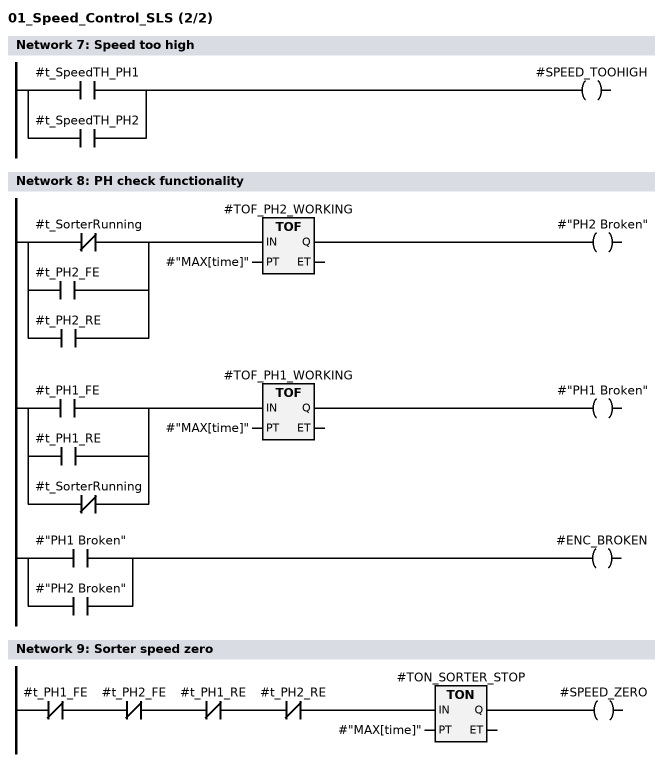
   RUNG wire#powerrail
      Contact( #t_SpeedTH_PH1 )
      wire#w1
      Coil( #SPEED_TOOHIGH )
   END_RUNG
   RUNG wire#powerrail
      Contact( #t_SpeedTH_PH2 )
   END_RUNG wire#w1
   // the same network as SCL:
   #SPEED_TOOHIGH := #t_SpeedTH_PH1 OR #t_SpeedTH_PH2;
END_REGION

REGION Network 8: PH check functionality
   #TOF_PH2_WORKING.TOF(IN := NOT #t_SorterRunning OR #t_PH2_FE OR #t_PH2_RE, PT := #"MAX[time]");
   #"PH2 Broken" := #TOF_PH2_WORKING.Q;
   #TOF_PH1_WORKING.TOF(IN := #t_PH1_FE OR #t_PH1_RE OR NOT #t_SorterRunning, PT := #"MAX[time]");
   #"PH1 Broken" := #TOF_PH1_WORKING.Q;
   #ENC_BROKEN := #"PH1 Broken" OR #"PH2 Broken";
END_REGION

REGION Network 9: Sorter speed zero
   #TON_SORTER_STOP.TON(IN := NOT #t_PH1_FE AND NOT #t_PH2_FE AND NOT #t_PH1_RE AND NOT #t_PH2_RE,
                        PT := #"MAX[time]");
   #SPEED_ZERO := #TON_SORTER_STOP.Q;
END_REGION
END_FUNCTION_BLOCK

FUNCTION "00_Only for Commissioning" : Void   // FC1, F_LAD
{ S7_Optimized_Access := 'TRUE' }
VERSION : 0.1
// Management of bypass to use during commissioning
BEGIN

REGION Network 1: Example
   // One network per node
   // TRUE if the node is not ready to be used
   // FALSE if the node is ready
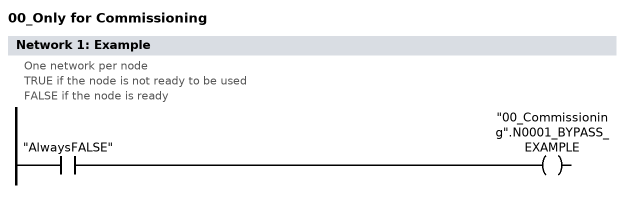
   RUNG wire#powerrail
      Contact( "AlwaysFALSE" )
      Coil( "00_Commissioning".N0001_BYPASS_EXAMPLE )
   END_RUNG
   // the same network as SCL:
   "00_Commissioning".N0001_BYPASS_EXAMPLE := "AlwaysFALSE";
END_REGION
END_FUNCTION

FUNCTION "01_Settings" : Void   // FC2, F_FBD
{ S7_Optimized_Access := 'TRUE' }
VERSION : 0.1
BEGIN

REGION Network 1: To be used in case of overall settings
   // for example in case of Tristate diagnostic
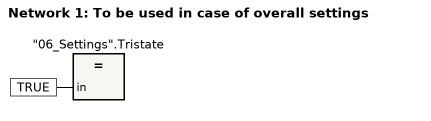
   "06_Settings".Tristate := TRUE;
END_REGION
END_FUNCTION

FUNCTION "02_EM Push Button" : Void   // FC3, F_LAD
{ S7_Optimized_Access := 'TRUE' }
VERSION : 0.1
BEGIN

REGION Network 1: One network per node
   // One FB2 per input module with E-Stop push button
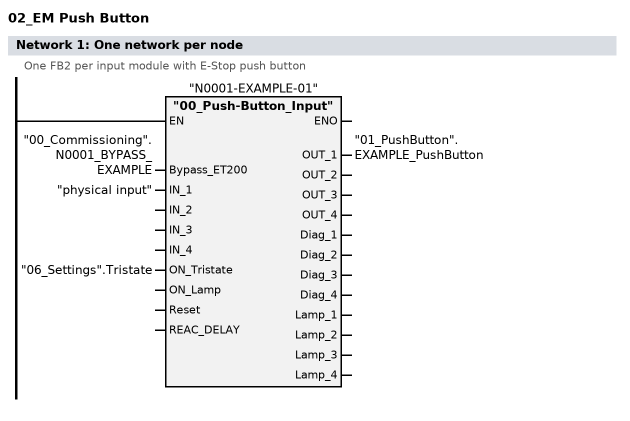
   RUNG wire#powerrail
      "N0001-EXAMPLE-01"(Bypass_ET200 := "00_Commissioning".N0001_BYPASS_EXAMPLE, IN_1 := "physical input", IN_2 :=, IN_3 :=, IN_4 :=, ON_Tristate := "06_Settings".Tristate, ON_Lamp :=, Reset :=, REAC_DELAY :=, OUT_1 => "01_PushButton".EXAMPLE_PushButton, OUT_2 =>, OUT_3 =>, OUT_4 =>, Diag_1 =>, Diag_2 =>, Diag_3 =>, Diag_4 =>, Lamp_1 =>, Lamp_2 =>, Lamp_3 =>, Lamp_4 =>)
   END_RUNG
   // the same network as SCL:
   "N0001-EXAMPLE-01"(Bypass_ET200 := "00_Commissioning".N0001_BYPASS_EXAMPLE,   // "00_Push-Button_Input"
                      IN_1 := "physical input",
                      ON_Tristate := "06_Settings".Tristate,
                      OUT_1 => "01_PushButton".EXAMPLE_PushButton);
END_REGION
END_FUNCTION

FUNCTION "03_Zone Cumulative" : Void   // FC4, F_FBD
{ S7_Optimized_Access := 'TRUE' }
VERSION : 0.1
BEGIN

REGION Network 1: One network per zone PB Com
   // Cumulative of the E-Stop Push buttons, based on the cause & effect matrix
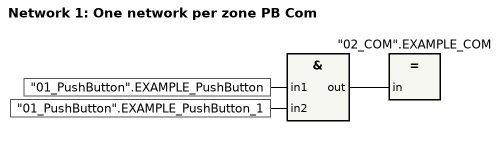
   "02_COM".EXAMPLE_COM := "01_PushButton".EXAMPLE_PushButton AND "01_PushButton".EXAMPLE_PushButton_1;
END_REGION
END_FUNCTION

FUNCTION "04_ESTOP" : Void   // FC5, F_FBD
{ S7_Optimized_Access := 'TRUE' }
VERSION : 0.1
// For each Sorter, repeat the first three networks
BEGIN

REGION Network 1: SORTER CONV
   // estop with 150ms delay for the ind lines
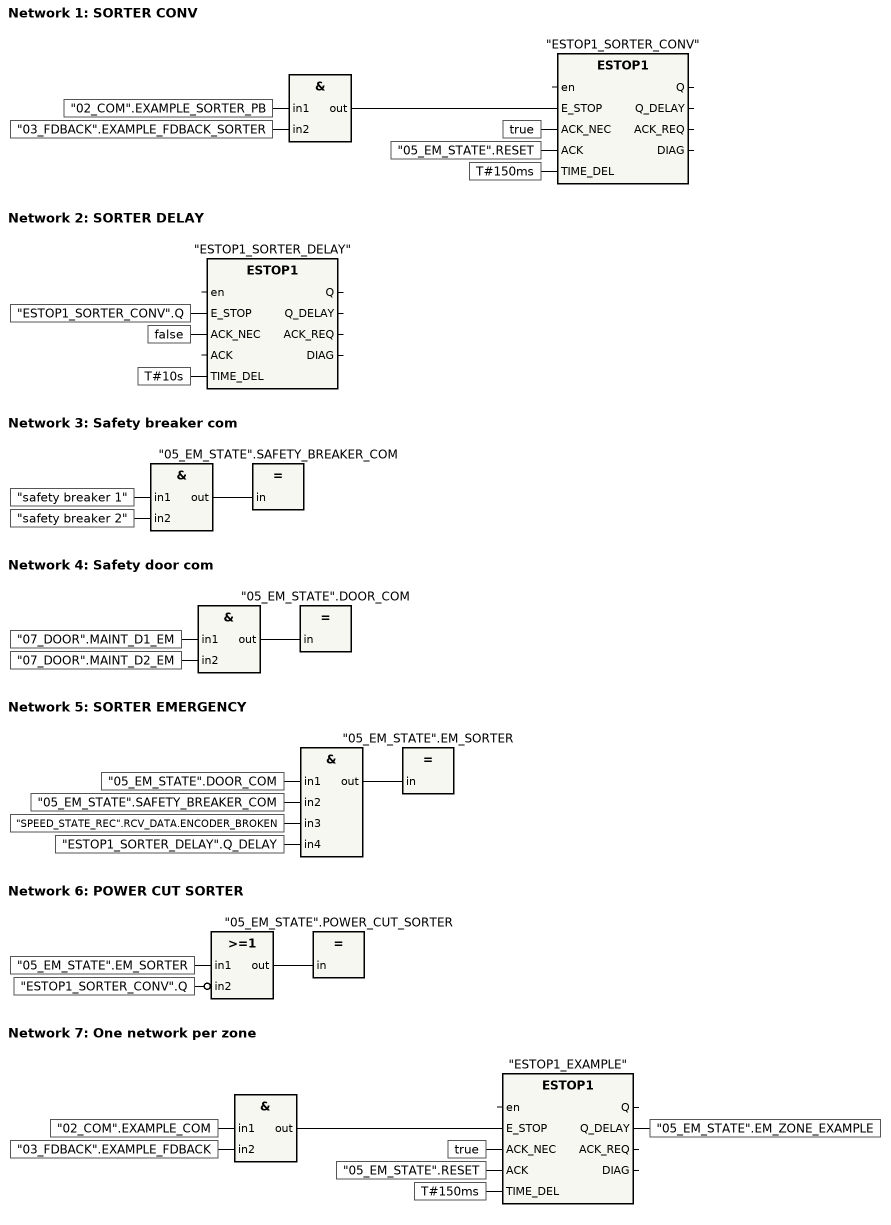
   "ESTOP1_SORTER_CONV"(E_STOP := "02_COM".EXAMPLE_SORTER_PB AND "03_FDBACK".EXAMPLE_FDBACK_SORTER,   // ESTOP1
                        ACK_NEC := true,
                        ACK := "05_EM_STATE".RESET,
                        TIME_DEL := T#150ms);
END_REGION

REGION Network 2: SORTER DELAY
   // estop with 10s delay for the sorter, the delay can be decreased, not increased
   "ESTOP1_SORTER_DELAY"(E_STOP := "ESTOP1_SORTER_CONV".Q, ACK_NEC := false, TIME_DEL := T#10s);   // ESTOP1
END_REGION

REGION Network 3: Safety breaker com
   "05_EM_STATE".SAFETY_BREAKER_COM := "safety breaker 1" AND "safety breaker 2";
END_REGION

REGION Network 4: Safety door com
   "05_EM_STATE".DOOR_COM := "07_DOOR".MAINT_D1_EM AND "07_DOOR".MAINT_D2_EM;
END_REGION

REGION Network 5: SORTER EMERGENCY
   // overall emergency state
   "05_EM_STATE".EM_SORTER := "05_EM_STATE".DOOR_COM AND "05_EM_STATE".SAFETY_BREAKER_COM AND "SPEED_STATE_REC".RCV_DATA.ENCODER_BROKEN AND "ESTOP1_SORTER_DELAY".Q_DELAY;
END_REGION

REGION Network 6: POWER CUT SORTER
   "05_EM_STATE".POWER_CUT_SORTER := "05_EM_STATE".EM_SORTER OR NOT "ESTOP1_SORTER_CONV".Q;
END_REGION

REGION Network 7: One network per zone
   // Each zone can be stopped by the pushbutton cumuative or the feedback error
   "ESTOP1_EXAMPLE"(E_STOP := "02_COM".EXAMPLE_COM AND "03_FDBACK".EXAMPLE_FDBACK,   // ESTOP1
                    ACK_NEC := true,
                    ACK := "05_EM_STATE".RESET,
                    TIME_DEL := T#150ms,
                    Q_DELAY => "05_EM_STATE".EM_ZONE_EXAMPLE);
END_REGION
END_FUNCTION

FUNCTION "05_Output Feedback" : Void   // FC6, F_FBD
{ S7_Optimized_Access := 'TRUE' }
VERSION : 0.1
   VAR_TEMP
      DU_EX : Bool;
      ISPC_EX : Bool;
      ZONE_EX : Bool;
   END_VAR
BEGIN

REGION Network 1: NETWORK_COMMMENT_1
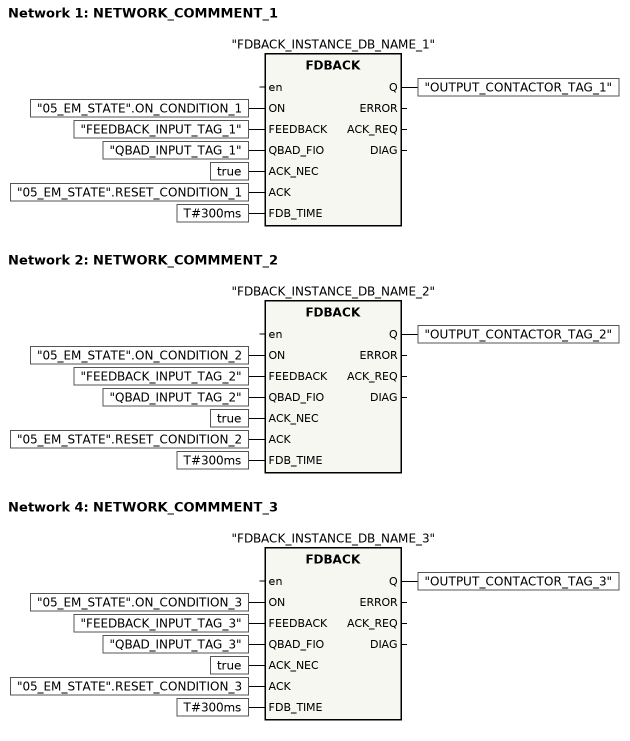
   "FDBACK_INSTANCE_DB_NAME_1"(ON := "05_EM_STATE".ON_CONDITION_1,   // FDBACK
                           FEEDBACK := "FEEDBACK_INPUT_TAG_1",
                           QBAD_FIO := "QBAD_INPUT_TAG_1",
                           ACK_NEC := true,
                           ACK := "05_EM_STATE".RESET_CONDITION_1,
                           FDB_TIME := T#300ms,
                           Q => "OUTPUT_CONTACTOR_TAG_1");
END_REGION

REGION Network 2: NETWORK_COMMMENT_2
   "FDBACK_INSTANCE_DB_NAME_2"(ON := "05_EM_STATE".ON_CONDITION_2,   // FDBACK
                           FEEDBACK := "FEEDBACK_INPUT_TAG_2",
                           QBAD_FIO := "QBAD_INPUT_TAG_2",
                           ACK_NEC := true,
                           ACK := "05_EM_STATE".RESET_CONDITION_2,
                           FDB_TIME := T#300ms,
                           Q => "OUTPUT_CONTACTOR_TAG_2");
END_REGION

REGION Network 4: NETWORK_COMMMENT_3
   "FDBACK_INSTANCE_DB_NAME_3"(ON := "05_EM_STATE".ON_CONDITION_3,   // FDBACK
                           FEEDBACK := "FEEDBACK_INPUT_TAG_3",
                           QBAD_FIO := "QBAD_INPUT_TAG_3",
                           ACK_NEC := true,
                           ACK := "05_EM_STATE".RESET_CONDITION_3,
                           FDB_TIME := T#300ms,
                           Q => "OUTPUT_CONTACTOR_TAG_3");
END_REGION
END_FUNCTION

FUNCTION "06_Feedback Error" : Void   // FC7, F_LAD
{ S7_Optimized_Access := 'TRUE' }
VERSION : 0.1
BEGIN

REGION Network 1: one network per node with safety output
   // use one FB4 for each output module with at least one drive unit, ISPC or zone controlled
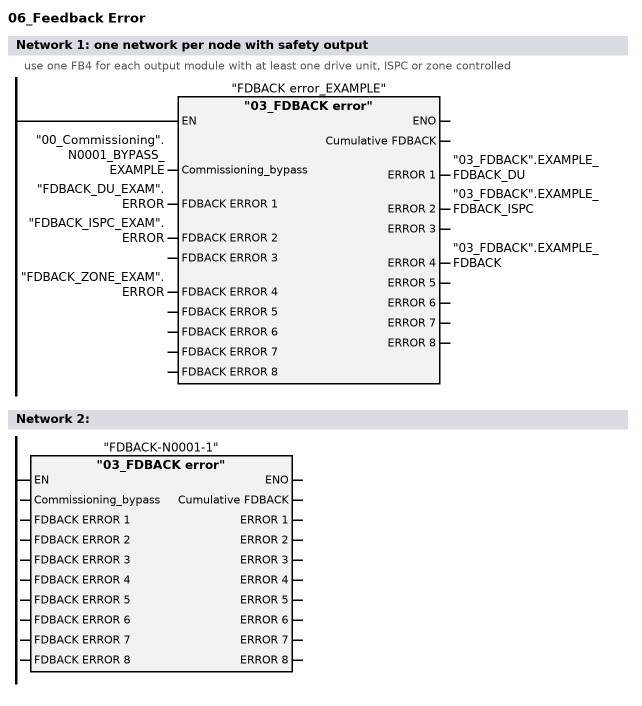
   RUNG wire#powerrail
      "FDBACK error_EXAMPLE"(Commissioning_bypass := "00_Commissioning".N0001_BYPASS_EXAMPLE, "FDBACK ERROR 1" := "FDBACK_DU_EXAM".ERROR, "FDBACK ERROR 2" := "FDBACK_ISPC_EXAM".ERROR, "FDBACK ERROR 3" :=, "FDBACK ERROR 4" := "FDBACK_ZONE_EXAM".ERROR, "FDBACK ERROR 5" :=, "FDBACK ERROR 6" :=, "FDBACK ERROR 7" :=, "FDBACK ERROR 8" :=, "Cumulative FDBACK" =>, "ERROR 1" => "03_FDBACK".EXAMPLE_FDBACK_DU, "ERROR 2" => "03_FDBACK".EXAMPLE_FDBACK_ISPC, "ERROR 3" =>, "ERROR 4" => "03_FDBACK".EXAMPLE_FDBACK, "ERROR 5" =>, "ERROR 6" =>, "ERROR 7" =>, "ERROR 8" =>)
   END_RUNG
   // the same network as SCL:
   "FDBACK error_EXAMPLE"(Commissioning_bypass := "00_Commissioning".N0001_BYPASS_EXAMPLE,   // "03_FDBACK error"
                          "FDBACK ERROR 1" := "FDBACK_DU_EXAM".ERROR,
                          "FDBACK ERROR 2" := "FDBACK_ISPC_EXAM".ERROR,
                          "FDBACK ERROR 4" := "FDBACK_ZONE_EXAM".ERROR,
                          "ERROR 1" => "03_FDBACK".EXAMPLE_FDBACK_DU,
                          "ERROR 2" => "03_FDBACK".EXAMPLE_FDBACK_ISPC,
                          "ERROR 4" => "03_FDBACK".EXAMPLE_FDBACK);
END_REGION

REGION Network 2
   RUNG wire#powerrail
      "FDBACK-N0001-1"(Commissioning_bypass :=, "FDBACK ERROR 1" :=, "FDBACK ERROR 2" :=, "FDBACK ERROR 3" :=, "FDBACK ERROR 4" :=, "FDBACK ERROR 5" :=, "FDBACK ERROR 6" :=, "FDBACK ERROR 7" :=, "FDBACK ERROR 8" :=, "Cumulative FDBACK" =>, "ERROR 1" =>, "ERROR 2" =>, "ERROR 3" =>, "ERROR 4" =>, "ERROR 5" =>, "ERROR 6" =>, "ERROR 7" =>, "ERROR 8" =>)
   END_RUNG
   // the same network as SCL:
   "FDBACK-N0001-1"();   // "03_FDBACK error"
END_REGION
END_FUNCTION

FUNCTION "07_Speed Control" : Void   // FC8, F_LAD
{ S7_Optimized_Access := 'TRUE' }
VERSION : 0.1
BEGIN

REGION Network 1: One network per sorter
END_REGION

REGION Network 2
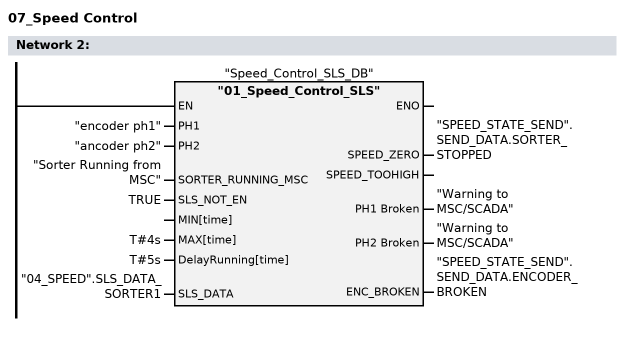
   RUNG wire#powerrail
      "Speed_Control_SLS_DB"(PH1 := "encoder ph1", PH2 := "ancoder ph2", SORTER_RUNNING_MSC := "Sorter Running from MSC", SLS_NOT_EN := TRUE, "MIN[time]" :=, "MAX[time]" := T#4s, "DelayRunning[time]" := T#5s, SLS_DATA := "04_SPEED".SLS_DATA_SORTER1, SPEED_ZERO => "SPEED_STATE_SEND".SEND_DATA.SORTER_STOPPED, SPEED_TOOHIGH =>, "PH1 Broken" => "Warning to MSC/SCADA", "PH2 Broken" => "Warning to MSC/SCADA", ENC_BROKEN => "SPEED_STATE_SEND".SEND_DATA.ENCODER_BROKEN)
   END_RUNG
   // the same network as SCL:
   "Speed_Control_SLS_DB"(PH1 := "encoder ph1",   // "01_Speed_Control_SLS"
                          PH2 := "ancoder ph2",
                          SORTER_RUNNING_MSC := "Sorter Running from MSC",
                          SLS_NOT_EN := TRUE,
                          "MAX[time]" := T#4s,
                          "DelayRunning[time]" := T#5s,
                          SLS_DATA := "04_SPEED".SLS_DATA_SORTER1,
                          SPEED_ZERO => "SPEED_STATE_SEND".SEND_DATA.SORTER_STOPPED,
                          "PH1 Broken" => "Warning to MSC/SCADA",
                          "PH2 Broken" => "Warning to MSC/SCADA",
                          ENC_BROKEN => "SPEED_STATE_SEND".SEND_DATA.ENCODER_BROKEN);
END_REGION
END_FUNCTION

FUNCTION "08_Gate Manager" : Void   // FC9, F_LAD
{ S7_Optimized_Access := 'TRUE' }
VERSION : 0.1
   VAR_TEMP
      temp_EXAMPLE_OPEN : Bool;
   END_VAR
BEGIN

REGION Network 1: Transfer Data from Speed Control
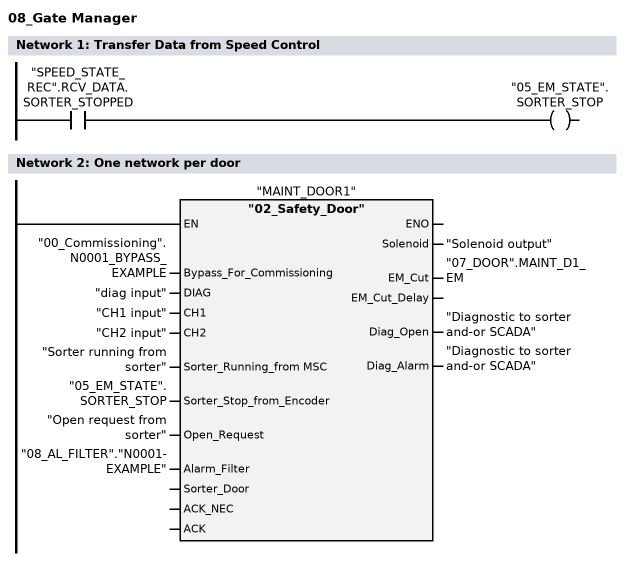
   RUNG wire#powerrail
      Contact( "SPEED_STATE_REC".RCV_DATA.SORTER_STOPPED )
      Coil( "05_EM_STATE".SORTER_STOP )
   END_RUNG
   // the same network as SCL:
   "05_EM_STATE".SORTER_STOP := "SPEED_STATE_REC".RCV_DATA.SORTER_STOPPED;
END_REGION

REGION Network 2: One network per door
   RUNG wire#powerrail
      "MAINT_DOOR1"(Bypass_For_Commissioning := "00_Commissioning".N0001_BYPASS_EXAMPLE, DIAG := "diag input", CH1 := "CH1 input", CH2 := "CH2 input", "Sorter_Running_from MSC" := "Sorter running from sorter", Sorter_Stop_from_Encoder := "05_EM_STATE".SORTER_STOP, Open_Request := "Open request from sorter", Alarm_Filter := "08_AL_FILTER"."N0001-EXAMPLE", Sorter_Door :=, ACK_NEC :=, ACK :=, Solenoid => "Solenoid output", EM_Cut => "07_DOOR".MAINT_D1_EM, EM_Cut_Delay =>, Diag_Open => "Diagnostic to sorter and-or SCADA", Diag_Alarm => "Diagnostic to sorter and-or SCADA")
   END_RUNG
   // the same network as SCL:
   "MAINT_DOOR1"(Bypass_For_Commissioning := "00_Commissioning".N0001_BYPASS_EXAMPLE,   // "02_Safety_Door"
                 DIAG := "diag input",
                 CH1 := "CH1 input",
                 CH2 := "CH2 input",
                 "Sorter_Running_from MSC" := "Sorter running from sorter",
                 Sorter_Stop_from_Encoder := "05_EM_STATE".SORTER_STOP,
                 Open_Request := "Open request from sorter",
                 Alarm_Filter := "08_AL_FILTER"."N0001-EXAMPLE",
                 Solenoid => "Solenoid output",
                 EM_Cut => "07_DOOR".MAINT_D1_EM,
                 Diag_Open => "Diagnostic to sorter and-or SCADA",
                 Diag_Alarm => "Diagnostic to sorter and-or SCADA");
END_REGION
END_FUNCTION

FUNCTION "00_Diagnostic PB" : Void   // FC10, STL
{ S7_Optimized_Access := 'TRUE' }
VERSION : 0.1
BEGIN

REGION Network 1: Example for coupler
   // each Push button has to be diagnosed, the output Q10005.0 is an example
         A     "01_PushButton".EXAMPLE_PushButton;
         O     "08_AL_FILTER"."N0001-EXAMPLE";
         =     "Tag_6";
END_REGION

REGION Network 2: Example for OPB
   // for each push button, use the following structure, the outputQ10005.0 is an example
         AN    "01_PushButton".EXAMPLE_PushButton;
         AN    "08_AL_FILTER"."N0001-EXAMPLE";
         =     "Tag_6";
END_REGION
END_FUNCTION

FUNCTION "01_DIagnostic Status" : Void   // FC11, STL
{ S7_Optimized_Access := 'TRUE' }
VERSION : 0.1
// Diagnostic for 
// sorter and zone status
// safety breaker status
BEGIN

REGION Network 1: Heartbeat
   // heartbeat sent to the Sorter Q0.0 is an example, normally the heartbeat is the first bit sent
         A     "Clock_0.5Hz";
         =     "Tag_3";
END_REGION

REGION Network 2: Sorter example
   // for each sorter, the ESTOP
   //SAFETYPLCEMERGENCYRE
         A     "ESTOP1_SORTER_CONV".Q;
         =     "Tag_1";

   //SAFETYPLCPOWERCUT
         A     "05_EM_STATE".POWER_CUT_SORTER;
         =     "Tag_4";
END_REGION

REGION Network 3: zone example
   // q10002.2  is an example
         A     "ESTOP1_EXAMPLE".Q;
         =     "Tag_5";
END_REGION

NETWORK
TITLE = Safety breaker
// Same logic as an E-STOP Push Button
END_FUNCTION

FUNCTION "02_Diagnostic Profinet" : Void   // FC12, LAD
{ S7_Optimized_Access := 'TRUE' }
VERSION : 0.1
   VAR_TEMP
      deviceState : Int;
      deviceState_1 : Int;
      deviceState_2 : Int;
      deviceState_3 : Int;
   END_VAR
BEGIN

REGION Network 1: MADA123 / One network per Subnet
   // LADDR:
   // You select the PROFINET IO or DP master system at the LADDR parameter by means of the hardware identifier.
   // 
   // The hardware identifier is available:
   // -Either in the Network view of the properties of the PROFINET IO or DP master system
   // -Or in the PLC tag table in the listed system constants with the data type HW_IOSYSTEM.
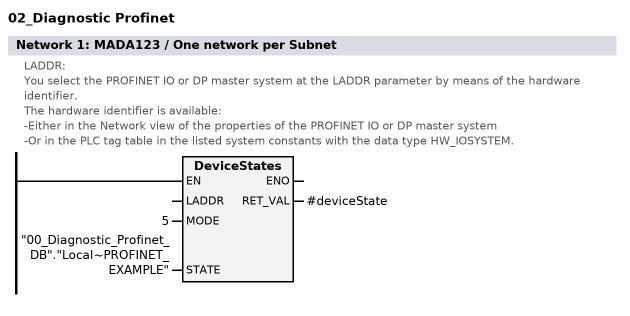
   // no SCL statement known for DeviceStates: written as a call
   #deviceState := DeviceStates(MODE := 5, STATE := "00_Diagnostic_Profinet_DB"."Local~PROFINET_EXAMPLE");
END_REGION
END_FUNCTION

FUNCTION "03_Diagnostic Nodes" : Void   // FC13, STL
{ S7_Optimized_Access := 'TRUE' }
VERSION : 0.1
BEGIN

REGION Network 1: One network per subnet
   // "00_Diagnostic_Profinet_DB"."Local~PROFINET_EXAMPLE"[x]
   // x = node number
   // 
   // Q10005.0 is an example
         AN    "00_Diagnostic_Profinet_DB"."Local~PROFINET_EXAMPLE"[1];
         =     "Tag_6";
         A     "00_Diagnostic_Profinet_DB"."Local~PROFINET_EXAMPLE"[1];
         =     "08_AL_FILTER"."N0001-EXAMPLE";
END_REGION
END_FUNCTION

FUNCTION "04_Diagnostic general alarms" : Void   // FC14, STL
{ S7_Optimized_Access := 'TRUE' }
VERSION : 0.1
// for other alarms diagnosed by the PLC
BEGIN
END_FUNCTION

FUNCTION "05_Diagnostic Feedback Error" : Void   // FC16, STL
{ S7_Optimized_Access := 'TRUE' }
VERSION : 0.1
BEGIN

REGION Network 1: Example
   // Each Feedbak error will be diagnosed in the same way as the Pushbuttons Q10005.0 is an example
         A     "03_FDBACK".EXAMPLE_FDBACK;
         =     "Tag_6";
END_REGION
END_FUNCTION

ORGANIZATION_BLOCK "Main"   // OB1, LAD, ProgramCycle
TITLE = "Main Program Sweep (Cycle)"
{ S7_Optimized_Access := 'TRUE' }
VERSION : 0.1
   VAR_INPUT
      Initial_Call : Bool;   // Initial call of this OB
      Remanence : Bool;   // =True, if remanent data are available
   END_VAR
BEGIN

REGION Network 1
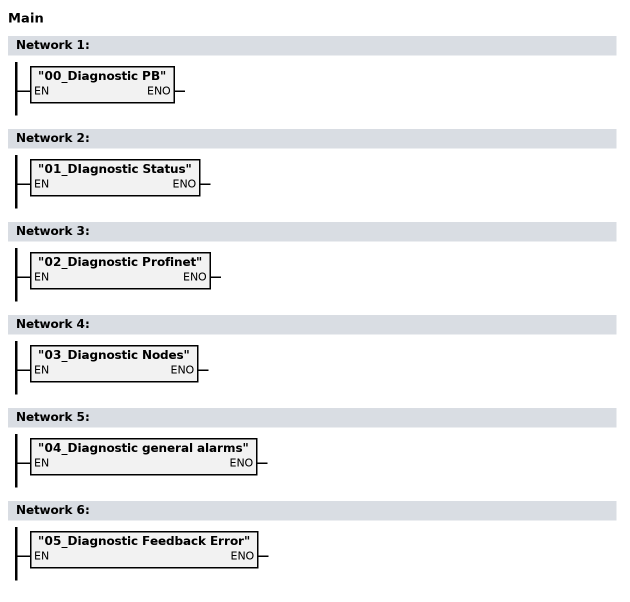
   RUNG wire#powerrail
      "00_Diagnostic PB"()
   END_RUNG
   // the same network as SCL:
   "00_Diagnostic PB"();
END_REGION

REGION Network 2
   RUNG wire#powerrail
      "01_DIagnostic Status"()
   END_RUNG
   // the same network as SCL:
   "01_DIagnostic Status"();
END_REGION

REGION Network 3
   RUNG wire#powerrail
      "02_Diagnostic Profinet"()
   END_RUNG
   // the same network as SCL:
   "02_Diagnostic Profinet"();
END_REGION

REGION Network 4
   RUNG wire#powerrail
      "03_Diagnostic Nodes"()
   END_RUNG
   // the same network as SCL:
   "03_Diagnostic Nodes"();
END_REGION

REGION Network 5
   RUNG wire#powerrail
      "04_Diagnostic general alarms"()
   END_RUNG
   // the same network as SCL:
   "04_Diagnostic general alarms"();
END_REGION

REGION Network 6
   RUNG wire#powerrail
      "05_Diagnostic Feedback Error"()
   END_RUNG
   // the same network as SCL:
   "05_Diagnostic Feedback Error"();
END_REGION
END_ORGANIZATION_BLOCK

ORGANIZATION_BLOCK "Programming error"   // OB121, LAD, ProgrammingError
{ S7_Optimized_Access := 'TRUE' }
VERSION : 0.1
   VAR_INPUT
      BlockNr : UInt;   // Number of causing block
      Reaction : USInt;   // 0:ignore, 1:substitute, 2:skip
      Fault_ID : Byte;   // Fault identifier
      BlockType : USInt;   // 16#01:OB, 16#02:FC, 16#03:FB, 16#04:SFC, 16#05:SFB, 16#06:DB: Type of block causing the error
      Area : USInt;   // Area where the error occured
      DBNr : DB_ANY;   // DB number if Area = DB or DI
      Csg_OBNr : OB_Any;   // Number of OB causing the error
      Csg_Prio : USInt;   // Priority of OB causing the error
      Width : USInt;   // 0:bit, 1:byte, 2:word, 3:dword, 4:lword
   END_VAR
BEGIN
END_ORGANIZATION_BLOCK

ORGANIZATION_BLOCK "IO access error"   // OB122, LAD, IOAccessError
{ S7_Optimized_Access := 'TRUE' }
VERSION : 0.1
   VAR_INPUT
      BlockNr : UInt;   // Number of causing block
      Reaction : USInt;   // 0:ignore, 1:substitute, 2:skip
      Fault_ID : Byte;   // 16#42:reading, 16#43:writing
      BlockType : USInt;   // 16#01:OB, 16#02:FC, 16#03:FB, 16#04:SFC, 16#05:SFB, 16#06:DB: Type of block causing the error
      Area : USInt;   // 16#81:I, 16#82:Q: IO area where the IOaccess error occured
      DBNr : DB_ANY;   // Reserved for system
      Csg_OBNr : OB_Any;   // Number of OB causing the error
      Csg_Prio : USInt;   // Priority of OB causing the error
      Width : USInt;   // 0:bit, 1:byte, 2:word, 3:dword, 4:lword
   END_VAR
BEGIN
END_ORGANIZATION_BLOCK

// folder: RTG_POST

FUNCTION "RTG2_POST" : Void   // FC15, LAD
{ S7_Optimized_Access := 'TRUE' }
VERSION : 0.1
BEGIN

REGION Network 1: Send the data to RTG1
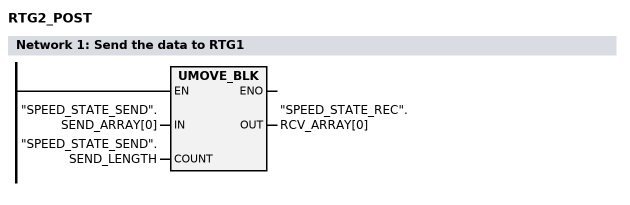
   UMOVE_BLK(IN := "SPEED_STATE_SEND".SEND_ARRAY[0],
             COUNT := "SPEED_STATE_SEND".SEND_LENGTH,
             OUT => "SPEED_STATE_REC".RCV_ARRAY[0]);
END_REGION
END_FUNCTION

FUNCTION "RTG1_POST" : Void   // FC17, LAD
{ S7_Optimized_Access := 'TRUE' }
VERSION : 0.1
BEGIN

REGION Network 1: Send the acknowledgment telegram to RTG2
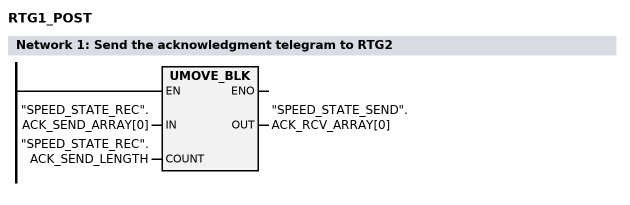
   UMOVE_BLK(IN := "SPEED_STATE_REC".ACK_SEND_ARRAY[0],
             COUNT := "SPEED_STATE_REC".ACK_SEND_LENGTH,
             OUT => "SPEED_STATE_SEND".ACK_RCV_ARRAY[0]);
END_REGION
END_FUNCTION